{attribute 'qualified_only'}
{attribute 'strict'}
{attribute 'to_string'}
TYPE eBA :
(
	MoveL 			:=0,
	MoveJ			:=1,
	MoveLRelativ 	:=2,
	MoveJRelativ 	:=3,
	SetDO			:=4,
	ReadDI			:=5,
	NavigateToGoal	:=7,
	NavigateToPoint	:=8,
	Dock			:=9,
	Undock			:=10,
	Home			:=11
	
);
END_TYPE

(* stored: Version 1.1.0.1, ProductVersion 3.1.4026.18
   DUT eBA: Id {229201d8-2c42-4601-b776-bb44db293d9d} *)
